FUNCTION FGetInstance : STRING
VAR_INPUT
	isample: I_BaseString;
END_VAR
VAR
END_VAR

FGetInstance := isample.GetString();

END_FUNCTION

(* stored: Version 1.1.0.1, ProductVersion 3.1.4024.3
   POU FGetInstance: Id {62980089-a5aa-4474-854e-0fc0ffc9faee}, SpecialFunc None *)
